// TIA Portal V20 export
DATA_BLOCK "Simulation_DB"   // DB139
// stored: InstanceOfName Unit1.Em5.Simulation, InstanceOfType FB, Namespace Unit1.Em5
"Unit1.Em5.Simulation"
   // VAR_INPUT
   //    simulation : Bool;
   // END_VAR
   // VAR
   //    Simulation_addon_Instance { S7_SetPoint := 'True'} : "Simulation_addon";
   //    Simulation_addon_Instance_1 { S7_SetPoint := 'True'} : "Simulation_addon";
   //    Simulation_addon_Instance_2 { S7_SetPoint := 'True'} : "Simulation_addon";
   //    Simulation_addon_Instance_3 { S7_SetPoint := 'True'} : "Simulation_addon";
   // END_VAR
BEGIN
END_DATA_BLOCK
